# EPICS substitutions: EUROTHRM/EUROTHRM-IOC-01App/Db/devEurothrmA03.substitutions
# Note: this file is generated by generate_substitutions.py
file devEurothrm.template {
pattern { P, GAD, LAD, MODBUS_PV, MODBUS_SP, MODBUS_P, MODBUS_I, MODBUS_D, MODBUS_HS, MODBUS_LS, MODBUS_AT, MODBUS_HO, MODBUS_OP }
{ "\$(P)", "0", "3", "2049", "2050", "2054", "2056", "2057", "2159", "2160", "2318", "2078", "2051" }
}
